FUNCTION_BLOCK FB_Valve_monitor
VAR_INPUT
	Coil_state:BOOL;
	Energise_to_open:BOOL;
	Valve_open:BOOL;
	Valve_closed:BOOL;
	Open_time:TIME;
	Close_time:TIME;
END_VAR
VAR_OUTPUT
	Not_opening:BOOL;
	Not_closing:BOOL;
	Open_and_closed:BOOL;
END_VAR
VAR
	TON_0: TON;
END_VAR

Valve_monitor();

METHOD Valve_monitor
VAR_INPUT
END_VAR
VAR_INST // added by the converter: edge detectors and wires of the graphical bodies
    _w1 : BOOL;
END_VAR
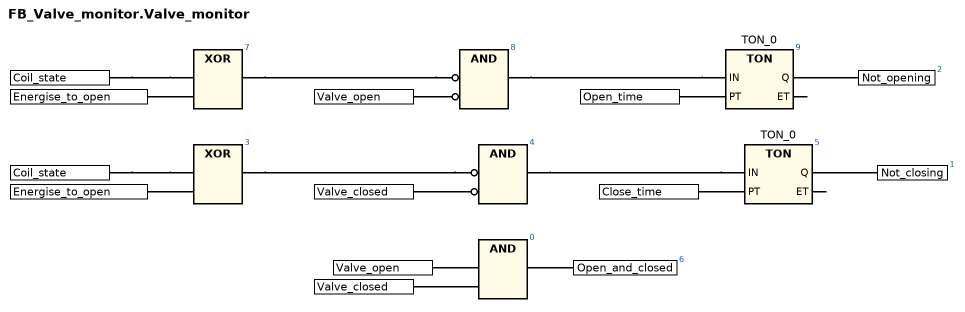
_w1 := Valve_open AND Valve_closed;
Not_closing := TON_0.Q;
Not_opening := TON_0.Q;
TON_0(IN := NOT (Coil_state XOR Energise_to_open) AND NOT Valve_closed, PT := Close_time); // TON
Open_and_closed := _w1;
TON_0(IN := NOT (Coil_state XOR Energise_to_open) AND NOT Valve_open, PT := Open_time); // TON
END_METHOD

END_FUNCTION_BLOCK

(* stored: Version 1.1.0.1, ProductVersion 3.1.4024.0
   POU FB_Valve_monitor: Id {31f1f1ef-fef2-4da7-a5d2-536c33690cbe}, SpecialFunc None
   Method Valve_monitor: Id {187782b6-0689-466b-ba3d-a7b3d461bc08} *)
